(* Logix 5000 project; controller QW361 vendor 1 type 14 code 107 rev 32.11; software revision 32.00; part 19 of 20 *)
(* tags used below, declared in another part *)
   ALM_ACK : BOOL;   // Alarm acknowledge
   alm_pwrup_done : BOOL;
   ALM_RESET : BOOL;   // Alarm reset
   ALM_TEST : BOOL;   // Alarm test
   analogfb_pwrup_done : BOOL;
   ATSFLT : ALM;   // ATS fault
   ATSGEN : ALM;   // ATS in generator
   BAND_B01_MAXSPD_LVL : REAL;   // Band 1 maximum speed level
   BAND_B01_MINSPD_LVL : REAL;   // Band 1 minimum speed level
   BAND_B01_START : REAL;   // Wet well level to start lead pump
   BAND_B01_STOP : REAL;   // Wet well level to stop lead pump
   BAND_B02_MAXSPD_LVL : REAL;   // band 2 maximum speed level
   BAND_B02_MINSPD_LVL : REAL;   // band 2 minimum speed level
   BAND_B02_START : REAL;   // Wet well level to start lag pump
   BAND_B02_STOP : REAL;   // Wet well level to stop lag pump
   BAND_CURRENT : DINT;   // Current band
   CRP : ALM;   // Control power failure
   DG1 : MOTOR;   // Diesel generator
   DG1_FL : ALM;   // Diesel generator fault alarm
   DG1BAT : ALM;   // Battery low / fail
   DG1LSL1 : ALM;   // Low fuel
   DG1LSL2 : ALM;   // Low oil
   DG1RUN : ALM;   // Diesel generator running
   Dialer : BOOL[256];
   DIALOUT_ON : BOOL;
   digitalnf_pwrup_done : BOOL;
   duty_pwrup_done : BOOL;
   FIT001 : PRANALOG;   // Station discharge flow
   FIT001_CA : ALM;   // Station discharge flow calibrate mode alarm
   FIT001_FL : ALM;   // Station discharge flow sensor fail alarm
   FIT001_hh : ALM;   // Station discharge flow high high alarm
   FIT001_hi : ALM;   // Station discharge flow high alarm
   FIT001_ll : ALM;   // Station discharge flow low low alarm
   FIT001_lo : ALM;   // Station discharge flow low alarm
   FROM_QW360 : COMMBLOCK;
   FunctionBlock_Cycle_Time : REAL;   // Main Task Cycle Time in mseconds
   HardwareFault : BOOL;   // System hardware fault
   HMI_time : DateTime;
   HMI_time_set : BOOL;
   Last_Minute : DINT;
   LIT001 : PRANALOG;   // Wet well level
   LIT001_CA : ALM;   // Wet well level calibrate mode alarm
   LIT001_FL : ALM;   // Wet well level sensor fail alarm
   LIT001_hh : ALM;   // Wet well level high high alarm
   LIT001_hi : ALM;   // Wet well level high alarm
   LIT001_ll : ALM;   // Wet well level low low alarm
   LIT001_lo : ALM;   // Wet well level low alarm
   LSH001 : ALM;   // Station high float
   LSH002 : ALM;   // Station hihi float
   main_comm_pwrup_done : BOOL;
   MainTask_Cycle_Time : REAL;   // Main Task Cycle Time in mseconds
   motor_pwrup_done : BOOL;
   P001 : MOTOR;   // Raw sewage pump 1
   P001_FL : ALM;   // Raw sewage pump 1 fault alarm
   P001_LK : BOOL;   // Raw sewage pump 1 leak
   P001_OL : BOOL;   // Raw sewage pump 1 overload
   P001_TMP : BOOL;   // Raw sewage pump 1 temp
   P001SP : ANALOGFB;   // Raw sewage pump 1 speed
   P001SP_FL : ALM;   // Raw sewage pump 1 speed control fail alarm
   P002 : MOTOR;   // Raw sewage pump 2
   P002_FL : ALM;   // Raw sewage pump 2 fault alarm
   P002_LK : BOOL;   // Raw sewage pump 2 leak
   P002_OL : BOOL;   // Raw sewage pump 2 overload
   P002_TMP : BOOL;   // Raw sewage pump 2 temp
   P002SP : ANALOGFB;   // Raw sewage pump 2 speed
   P002SP_FL : ALM;   // Raw sewage pump 2 speed control fail alarm
   P00x : DUTY;   // Raw sewage pump duty
   P00xXA1 : ALM;   // Single raw sewage pump unavailable
   P00xXA2 : ALM;   // Multiple raw sewage pump unavailable
   pid_pwrup_done : BOOL;
   pranalog_pwrup_done : BOOL;
   pwrdown_time : DINT;
   report_pwrup_done : BOOL;
   sequence_pwrup_done : BOOL;
   SoftwareFault : BOOL;   // System software fault
   TO_QW360 : COMMBLOCK;
   valve_pwrup_done : BOOL;
   WALLCLOCK : DateTime;   // Global date / time
   WALLCLOCK_lock : BOOL;
   Watchdog_Relay : BOOL;
   XAFLOAT : ALM;   // Station in float mode
   XAHWARE : ALM;   // PLC hardware fault
   XASWARE : ALM;   // PLC software fault

PROGRAM AlmProgram   (* main routine Alms *)
VAR
   alm : ALM := (enmn := 1, enau := 1, alarm_tonr.TimerEnable := 1, alarm_tonr.Reset := 1);
   bit_num : DINT := 256;
   channel_num : DINT := 257;
   Controller_Status : DINT := 12640;
   Dint_Bit : DINT := 31;
   Dint_Word : DINT := 7;
   fail_pending : BOOL;
   Faulty_Modules : DINT := 3;
   latched_alarm : BOOL;
   num_channels : DINT := 256;
   temp_array : BOOL[256];
END_VAR

ROUTINE AlmRoutine   (* structured text *)
   SBR(alm);
   
   (* Alm function block *)
   
   (* Does all control processing for alarms *)
   
   (* Calling parameters: *)
   (*     alm : ALM *)
   
   (* Globals used: *)
   
   (* Globals changed: *)
   (*     fail_pending *)
   
   (*-------------------------------------------------------------------------------------------------------------------------------------------------*)
   //alm.enmn := 1;
   
   (* Load fault time with preset value *)
   alm.alarm_tonr.PRE := alm.dlay * 1000;
   alm.alarm_tonr.TimerEnable := 1;
   
   (* handle the alarms and events outputs *)
   
   (* check for previously latched alarms *)
   latched_alarm := alm.alarm AND alm.latch AND NOT alm.reset;
   
   (* calculate the fail pending *)
   IF
           NOT alm.enau
       OR
           NOT alm.enmn
       OR
           NOT alm.raw AND NOT latched_alarm
   
   THEN
       fail_pending := 0;
   
   ELSE
       fail_pending := 1;
   END_IF;
   
   (* time the fail pending *)
   alm.alarm_tonr.Reset := NOT fail_pending;
   TONR(alm.alarm_tonr);
   
   (* get the output *)
   alm.alarm := alm.alarm_tonr.DN;
   
   (* turn on the alarm channel if this is in alarm *)
   IF alm.alarm AND alm.chan > 0 AND alm.chan <= num_channels THEN
       temp_array[alm.chan - 1] := 1;
   END_IF;
   
   (* reset mometaries *)
   IF alm.reset THEN alm.reset := 0; END_IF;
   
   RET(alm);
   
END_ROUTINE

ROUTINE Alms   (* structured text *)
   (* Alm processing program *)
   
   (* Does all basic processing for all alms by calling the alm function block for each *)
   
   (* Globals used: *)
   
   (* Globals changed: *)
   (*     alm_pwrup_done *)
   
   (*-------------------------------------------------------------------------------------------------------------------------------------------------*)
   
   
   (* clear the channel array *)
   
   (* get the size of the channel array *)
   num_channels := 256;
   
   (* now clear the entire array *)
   FOR channel_num := 1 TO num_channels DO
       temp_array[channel_num - 1] := 0;
   END_FOR;
   
   
   (* get the fault records *)
   GSV( MODULE, , ledstatus, Faulty_Modules );
   GSV(CONTROLLERDEVICE, , STATUS, Controller_Status );
   
   (* hardware fault if the IO light is neither solid on or off OR major fault or minor fault unrecoverable *)
   HardwareFault := ((Faulty_Modules <> 3) AND (Faulty_Modules <> 0)) OR ((Controller_Status AND 16#F00) <> 0);
   
   (* software fault if the unit is not in run mode (includes unrecoverable faults) *)
   SoftwareFault := (Controller_Status AND 16#FF) <> 16#60;
   
   
   (************ insert alms here ***************)
   
   (* 1.  Call the discrete alarms *)
   JSR (Discretes);
   
   (* 2.  Call the motor alarms *)
   JSR (Motors);
   
   (* 3.  Call the valve alarms *)
   JSR (Valves);
   
   (* 4.  Call the pranalog alarms *)
   JSR (Pranalogs);
   
   (* 5.  Call the Analogfb alarms *)
   JSR (Analogfbs);
   
   
   (* XAHWARE PLC Hardware fault *)
   
   (* process the inputs *)
   XAHWARE.raw := HardwareFault;
   XAHWARE.enau := 1;
   
   (* process the alarm *)
   JSR( AlmRoutine, 1, XAHWARE, XAHWARE );
   
   
   (* XASWARE PLC Software fault *)
   
   (* process the inputs *)
   XASWARE.raw := SoftwareFault;
   XASWARE.enau := 1;
   
   (* process the alarm *)
   JSR( AlmRoutine, 1, XASWARE, XASWARE );
   
   
   (* now copy the results from the temp array to the permanent array *)
   DIALOUT_ON := 0;
   FOR bit_num := 0 to 255 DO
   	Dint_Word := bit_num / 32;
   	Dint_Bit := bit_num - (Dint_Word * 32);
   	Dialer[bit_num] := temp_array[bit_num];
   	TO_QW360.ALMDINTS[Dint_Word].[Dint_Bit] := temp_array[bit_num];
   	IF Dialer[bit_num] THEN
   		DIALOUT_ON := 1;
   	END_IF;
   END_FOR;
   
   
   (* flag that powerup is done *)
   alm_pwrup_done := 1;
   
   
END_ROUTINE

ROUTINE Analogfbs   (* structured text *)
   (* P001SP_FL Raw sewage pump 1 speed control fail alarm *)
   
   (* process the inputs *)
   P001SP_FL.raw := P001SP_FL.raw;
   P001SP_FL.enau := 1;
   
   (* process the alarm *)
   JSR( AlmRoutine, 1, P001SP_FL, P001SP_FL );
   
   
   (* P002SP_FL Raw sewage pump 2 speed control fail alarm *)
   
   (* process the inputs *)
   P002SP_FL.raw := P002SP_FL.raw;
   P002SP_FL.enau := 1;
   
   (* process the alarm *)
   JSR( AlmRoutine, 1, P002SP_FL, P002SP_FL );
END_ROUTINE

ROUTINE Discretes   (* structured text *)
   
   (* CRP Control power failure *)
   
   (* process the inputs *)
   CRP.raw := CRP.raw;
   CRP.enau := 1;
   
   (* process the alarm *)
   JSR( AlmRoutine, 1, CRP, CRP );
   
   
   (* LS001 Station high float *)
   
   (* process the inputs *)
   LSH001.raw := LSH001.raw;
   LSH001.enau := 1;
   
   (* process the alarm *)
   JSR( AlmRoutine, 1, LSH001, LSH001 );
   
   
   (* LS002 Station hihi float *)
   
   (* process the inputs *)
   LSH002.raw := LSH002.raw;
   LSH002.enau := 1;
   
   (* process the alarm *)
   JSR( AlmRoutine, 1, LSH002, LSH002 );
   
   
   (* XAFLOAT Station in float mode *)
   
   (* process the inputs *)
   XAFLOAT.raw := XAFLOAT.raw;
   XAFLOAT.enau := 1;
   
   (* process the alarm *)
   JSR( AlmRoutine, 1, XAFLOAT, XAFLOAT );
   
   
   (* DG1LSL1 Low fuel *)
   
   (* process the inputs *)
   DG1LSL1.raw := DG1LSL1.raw;
   DG1LSL1.enau := 1;
   
   (* process the alarm *)
   JSR( AlmRoutine, 1, DG1LSL1, DG1LSL1 );
   
   
   (* DG1LSL2 Low oil *)
   
   (* process the inputs *)
   DG1LSL2.raw := DG1LSL2.raw;
   DG1LSL2.enau := 1;
   
   (* process the alarm *)
   JSR( AlmRoutine, 1, DG1LSL2, DG1LSL2 );
   
   
   (* DG1BAT Battery low / fail *)
   
   (* process the inputs *)
   DG1BAT.raw := DG1BAT.raw;
   DG1BAT.enau := 1;
   
   (* process the alarm *)
   JSR( AlmRoutine, 1, DG1BAT, DG1BAT );
   
   
   (* DG1RUN Diesel generator running *)
   
   (* process the inputs *)
   DG1RUN.raw := DG1.run_sts;
   DG1RUN.enau := 1;
   
   (* process the alarm *)
   JSR( AlmRoutine, 1, DG1RUN, DG1RUN );
   
   
   (* ATSGEN ATS in generator *)
   
   (* process the inputs *)
   ATSGEN.raw := ATSGEN.raw;
   ATSGEN.enau := 1;
   
   (* process the alarm *)
   JSR( AlmRoutine, 1, ATSGEN, ATSGEN );
   
   
   (* ATSFLT ATS fault *)
   
   (* process the inputs *)
   ATSFLT.raw := ATSFLT.raw;
   ATSFLT.enau := 1;
   
   (* process the alarm *)
   JSR( AlmRoutine, 1, ATSFLT, ATSFLT );
   
   
   (* P00xXA1 Single raw sewage pump unavailable *)
   
   (* process the inputs *)
   P00xXA1.raw := P00xXA1.raw;
   P00xXA1.enau := 1;
   
   (* process the alarm *)
   JSR( AlmRoutine, 1, P00xXA1, P00xXA1 );
   
   
   (* P00xXA2 Multiple raw sewage pump unavailable *)
   
   (* process the inputs *)
   P00xXA2.raw := P00xXA2.raw;
   P00xXA2.enau := 1;
   
   (* process the alarm *)
   JSR( AlmRoutine, 1, P00xXA2, P00xXA2 );
   
   
   
   
END_ROUTINE

ROUTINE Motors   (* structured text *)
   (* P001_FL Raw sewage pump 1 fault alarm *)
   
   (* process the inputs *)
   P001_FL.raw := P001_FL.raw;
   P001_FL.enau := 1;
   
   (* process the alarm *)
   JSR( AlmRoutine, 1, P001_FL, P001_FL );
   
   
   (* P002_FL Raw sewage pump 2 fault alarm *)
   
   (* process the inputs *)
   P002_FL.raw := P002_FL.raw;
   P002_FL.enau := 1;
   
   (* process the alarm *)
   JSR( AlmRoutine, 1, P002_FL, P002_FL );
   
   
   (* DG1_FL Diesel generator fault alarm *)
   
   (* process the inputs *)
   DG1_FL.raw := DG1_FL.raw;
   DG1_FL.enau := 1;
   
   (* process the alarm *)
   JSR( AlmRoutine, 1, DG1_FL, DG1_FL );
END_ROUTINE

ROUTINE Pranalogs   (* structured text *)
   (* LIT001_hi Wet well level high alarm *)
   
   (* process the inputs *)
   LIT001_hi.raw := LIT001_hi.raw;
   LIT001_hi.enau := 1;
   
   (* process the alarm *)
   JSR( AlmRoutine, 1, LIT001_hi, LIT001_hi );
   
   
   (* LIT001_lo Wet well level low alarm *)
   
   (* process the inputs *)
   LIT001_lo.raw := LIT001_lo.raw;
   LIT001_lo.enau := 1;
   
   (* process the alarm *)
   JSR( AlmRoutine, 1, LIT001_lo, LIT001_lo );
   
   
   (* LIT001_hh Wet well level high high alarm *)
   
   (* process the inputs *)
   LIT001_hh.raw := LIT001_hh.raw;
   LIT001_hh.enau := 1;
   
   (* process the alarm *)
   JSR( AlmRoutine, 1, LIT001_hh, LIT001_hh );
   
   
   (* LIT001_ll Wet well level low low alarm *)
   
   (* process the inputs *)
   LIT001_ll.raw := LIT001_ll.raw;
   LIT001_ll.enau := 1;
   
   (* process the alarm *)
   JSR( AlmRoutine, 1, LIT001_ll, LIT001_ll );
   
   
   (* LIT001_CA Wet well level calibrate mode alarm *)
   
   (* process the inputs *)
   LIT001_CA.raw := LIT001_CA.raw;
   LIT001_CA.enau := 1;
   
   (* process the alarm *)
   JSR( AlmRoutine, 1, LIT001_CA, LIT001_CA );
   
   
   (* LIT001_FL Wet well level sensor fail alarm *)
   
   (* process the inputs *)
   LIT001_FL.raw := LIT001_FL.raw;
   LIT001_FL.enau := 1;
   
   (* process the alarm *)
   JSR( AlmRoutine, 1, LIT001_FL, LIT001_FL );
   
   
   (* FIT001_hi Station discharge flow high alarm *)
   
   (* process the inputs *)
   FIT001_hi.raw := FIT001_hi.raw;
   FIT001_hi.enau := 1;
   
   (* process the alarm *)
   JSR( AlmRoutine, 1, FIT001_hi, FIT001_hi );
   
   
   (* FIT001_lo Station discharge flow low alarm *)
   
   (* process the inputs *)
   FIT001_lo.raw := FIT001_lo.raw;
   FIT001_lo.enau := 1;
   
   (* process the alarm *)
   JSR( AlmRoutine, 1, FIT001_lo, FIT001_lo );
   
   
   (* FIT001_hh Station discharge flow high high alarm *)
   
   (* process the inputs *)
   FIT001_hh.raw := FIT001_hh.raw;
   FIT001_hh.enau := 1;
   
   (* process the alarm *)
   JSR( AlmRoutine, 1, FIT001_hh, FIT001_hh );
   
   
   (* FIT001_ll Station discharge flow low low alarm *)
   
   (* process the inputs *)
   FIT001_ll.raw := FIT001_ll.raw;
   FIT001_ll.enau := 1;
   
   (* process the alarm *)
   JSR( AlmRoutine, 1, FIT001_ll, FIT001_ll );
   
   
   (* FIT001_CA Station discharge flow calibrate mode alarm *)
   
   (* process the inputs *)
   FIT001_CA.raw := FIT001_CA.raw;
   FIT001_CA.enau := 1;
   
   (* process the alarm *)
   JSR( AlmRoutine, 1, FIT001_CA, FIT001_CA );
   
   
   (* FIT001_FL Station discharge flow sensor fail alarm *)
   
   (* process the inputs *)
   FIT001_FL.raw := FIT001_FL.raw;
   FIT001_FL.enau := 1;
   
   (* process the alarm *)
   JSR( AlmRoutine, 1, FIT001_FL, FIT001_FL );
   
END_ROUTINE

ROUTINE Valves   (* structured text *)
   
END_ROUTINE
END_PROGRAM

PROGRAM AnalogfbProgram   (* main routine Analogfbs *)
VAR
   analogfb : ANALOGFB := (remote := 1, permit := 1, fail_tonr.TimerEnable := 1, fail_tonr.Reset := 1);
   fail_pending : BOOL;
   pwrup_dlayd : FBD_TIMER := (TimerEnable := 1, PRE := 10000, ACC := 10000, EN := 1, DN := 1);
END_VAR

ROUTINE AnalogfbRoutine   (* structured text *)
   SBR(analogfb);
   
   (* Analogfb function block *)
   
   (* Does all control processing for analog devices with feedback *)
   
   (* Calling parameters: *)
   (*     analogfb : ANALOGFB *)
   
   (* Globals used: *)
   (*     pwrup_dlayd *)
   
   (* Globals changed: *)
   (*     fail_pending *)
   
   (*-------------------------------------------------------------------------------------------------------------------------------------------------*)
   
   
   (* handle the failure logic first *)
   
   (* calculate the fail pending *)
   IF
           NOT analogfb.remote
       OR
   	    ( ABS( analogfb.out - analogfb.feedback ) <= 5.0 )
   	OR
   	    NOT pwrup_dlayd.DN
   THEN
       fail_pending := 0;
   ELSE
       fail_pending := 1;
   END_IF;
   
   (* time the fail pending *)
   analogfb.fail_tonr.PRE := analogfb.fail_dlay * 1000;
   analogfb.fail_tonr.TimerEnable := 1;
   analogfb.fail_tonr.Reset := NOT fail_pending;
   tonr(analogfb.fail_tonr);
   
   (* calculate the fail and clear if we're not in remote or we just powered up *)
   analogfb.fail := ( analogfb.fail AND ( NOT analogfb.fail_reset AND analogfb.remote AND pwrup_dlayd.DN ) ) OR analogfb.fail_tonr.DN;
   
   
   (* make the feedback *)
   IF analogfb.feedback_raw < 2 THEN
   	analogfb.feedback := 0;
   ELSIF analogfb.feedback_raw > 98 THEN
   	analogfb.feedback := 100;
   ELSE
   	analogfb.feedback := analogfb.feedback_raw;
   END_IF;
   
   
   (* handle the analog fb outputs *)
   
   (* if we're not permitted to control or not in remote or just powered up, set output to current feedback *)
   IF NOT analogfb.permit OR NOT analogfb.remote OR NOT pwrup_dlayd.DN THEN
   	analogfb.out := analogfb.feedback;
   
   (* if we're not in auto, set the output to the manual setpoint and track with the auto setpoint *)
   ELSIF NOT analogfb.auto THEN
   	analogfb.out := analogfb.out_man;
   
   (* otherwise, set the output to the auto setpoint and track with the manual setpoint*)
   ELSE
   	analogfb.out := analogfb.out_auto;
   END_IF;
   
   (* make sure both setpoints track *)
   analogfb.out_man := analogfb.out;
   analogfb.out_auto:= analogfb.out;
   
   
   (* process the momentary resets *)
   
   (* set the momentary resets equal to the current state *)
   IF analogfb.fail_reset THEN analogfb.fail_reset := 0; END_IF;
   
   RET(analogfb);
END_ROUTINE

ROUTINE Analogfbs   (* structured text *)
   (* Analogfb processing program *)
   
   (* Does all basic processing for all analogfbs by setting up inputs then calling the analogfb function block for each *)
   
   (* Globals used: *)
   
   (* Globals changed: *)
   (*     analogfb_pwrup_done *)
   (*     pwrup_dlayd *)
   (*     each analogfb *)
   
   (*-------------------------------------------------------------------------------------------------------------------------------------------------*)
   
   
   (* use a TONR to delay ac power recovery *)
   
   pwrup_dlayd.Reset := not analogfb_pwrup_done;
   TONR(pwrup_dlayd);
   
   
   (* process each analogfb as follows: (note these comments are only shown here for brevity) *)
   (*     1. set up inputs (specific to each analogfb and commented *)
   (*     2. call the analogfb processing function block *)
   (*     3. clear the momentary inputs if they were on *)
   (*     4. get the outputs *)
   
   
   (************ insert analogfbs here ***************)
   
   
   (* P001SP Raw sewage pump 1 speed *)
   
   (* set up the inputs *)
   P001SP.remote := 1;
   P001SP.permit := 1;
   P001SP.feedback_raw := P001SP.out;
   
   (* process the analog with feedback and reset the momentaries *)
   JSR( AnalogfbRoutine, 1, P001SP, P001SP );
   P001SP_FL.raw := P001SP.fail;
   
   
   (* P002SP Raw sewage pump 2 speed *)
   
   (* set up the inputs *)
   P002SP.remote := 1;
   P002SP.permit := 1;
   P002SP.feedback_raw := P002SP.out;
   
   (* process the analog with feedback and reset the momentaries *)
   JSR( AnalogfbRoutine, 1, P002SP, P002SP );
   P002SP_FL.raw := P002SP.fail;
   
   
   
   (* flag that powerup is done *)
   analogfb_pwrup_done := 1;
   
END_ROUTINE
END_PROGRAM

PROGRAM Communication   (* main routine Main_Comm *)
VAR
   bit_num : DINT := 256;
   WD_in : DINT := 6947;
   WD_out : DINT := 6947;
END_VAR

ROUTINE Main_Comm   (* structured text *)
   (* Message routine for communication from PLC to PLC *)
   
   (* Globals used: *)
   
   (* Globals changed: *)
   
   (*-------------------------------------------------------------------------------------------------------------------------------------------------*)
   
   
   (************ insert comm stuff here ***************)
   (* send data to Youngs Cove WWTP *)
   
   (* Plant PLC COMMS *)
   (* Monitor / Control the WatchDog from QW360.  This side is the slave side, we recieve a watchdog
   	number and loop it back.  If the number we read fails to change then communications has failed.
   	Once we get an new number it's ok. *)
   IF TO_QW360.WATCHDOG <> FROM_QW360.WATCHDOG THEN
   //	XA_LLCOMM.Raw := 0;
   	TO_QW360.WATCHDOG := FROM_QW360.WATCHDOG;
   ELSE
   //	XA_LLCOMM.Raw := 1;
   END_IF;
   
   
   (* Output Block to Plant PLC *)
   	(* Watchdog - done above *)
   	(* BOOLS *)
   	TO_QW360.BOOLS[0] := DIALOUT_ON; //dialer zone is active
   
   	(* INTEGERS *)
   	TO_QW360.DINTS[0] := 0;
   
   	(* REALS *)
   	TO_QW360.REALS[0] := LIT001.value;
   	TO_QW360.REALS[1] := FIT001.value;
   
   
   
   
   (* Input Block From Tower PLC *)
   	(* Watchdog - done above *)
   	(* BOOLS *)
   // := FROM_QW360.BOOLS[0];
   
   	(* INTEGERS *)
   // := FROM_QW360.DINTS[0];
   
   	(* REALS *)
   // := FROM_QW360.REALS[0]; //
   
   	(* ALARMS *)
   // Used directly in Alms subroutine;
   
   
   (* flag that powerup is done *)
   main_comm_pwrup_done := 1;
   
END_ROUTINE
END_PROGRAM

PROGRAM CycleTime   (* main routine MainRoutine *)
VAR
   cycle_timer1 : FBD_TIMER := (TimerEnable := 1, Reset := 1, ACC := 500, EN := 1, DN := 1);
   cycle_timer2 : FBD_TIMER := (TimerEnable := 1, EN := 1, TT := 1);
   cycle_timer3 : FBD_TIMER := (TimerEnable := 1);
   DATETIME_TEMP : DateTime := (Year := 2022, Month := 5, Day := 3, Hour := 16, Minute := 29, Second := 58, Microsecond := 621793, DayOfWeek := 2, DST_ON := 1);
   DOW_Century : DINT := 20;   // Century or upper two digits from the year
   DOW_Day : DINT := 3;   // Day of the Month 1-31
   DOW_Month : DINT := 3;   // Month 1 = March, 10=december, 11=Jan and 12=Feb
   DOW_Output : DINT := 2;   // Day of Week 0 = Sun, 1=Mon, 2=Tues, 3=Wed, 4=Thur, 5=Fri, 6=Sat
   DOW_Temp00 : REAL := 20.22;   // Intermediate Math Value
   DOW_Temp01 : REAL := 7.7999997;   // Intermediate Math Value
   DOW_Temp02 : REAL := 7.600001;   // Intermediate Math Value
   DOW_Temp03 : DINT := 7;   // Intermediate Math Value
   DOW_Temp04 : DINT := 40;   // Intermediate Math Value
   DOW_Temp05 : REAL := 5.5;   // Intermediate Math Value
   DOW_Temp06 : DINT := 5;   // Intermediate Math Value
   DOW_Temp07 : REAL := 5.0;   // Intermediate Math Value
   DOW_Temp08 : DINT := 5;   // Intermediate Math Value
   DOW_Temp09 : REAL := 10.0;   // Intermediate Math Value
   DOW_Temp10 : REAL := -30.0;   // Intermediate Math Value
   DOW_Temp11 : REAL := -8.0;   // Intermediate Math Value
   DOW_Temp12 : REAL := -3.0;   // Intermediate Math Value
   DOW_Temp13 : REAL := 2.0;   // Intermediate Math Value
   DOW_Temp14 : REAL := 2.0;   // Intermediate Math Value
   DOW_Temp15 : REAL := 2.0;   // Intermediate Math Value
   DOW_Year : DINT := 22;   // Year within the century or last two digits in year
END_VAR

ROUTINE CycleTime   (* structured text *)
   (* determine elapsed time of this task since last execution using three timers *)
   
   (* get the three timers elapsed time *)
   (* note one timer is resetting and the other two are timing *)
   TONR(cycle_timer1);
   TONR(cycle_timer2);
   TONR(cycle_timer3);
   
   (* of course, grab the output from the timer that was reset two cycles ago and add in any powerdown time *)
   IF cycle_timer1.Reset THEN
       MainTask_Cycle_Time := cycle_timer2.ACC + pwrdown_time;
   	cycle_timer1.Reset := 0;
   	cycle_timer2.Reset := 1;
   	cycle_timer3.Reset := 0;
   ELSIF cycle_timer2.Reset THEN
       MainTask_Cycle_Time := cycle_timer3.ACC + pwrdown_time;
   	cycle_timer1.Reset := 0;
   	cycle_timer2.Reset := 0;
   	cycle_timer3.Reset := 1;
   ELSE
       MainTask_Cycle_Time := cycle_timer1.ACC + pwrdown_time;
   	cycle_timer1.Reset := 1;
   	cycle_timer2.Reset := 0;
   	cycle_timer3.Reset := 0;
   END_IF;
   
   
   
   
END_ROUTINE

ROUTINE DayOfWeek   (* ladder *)
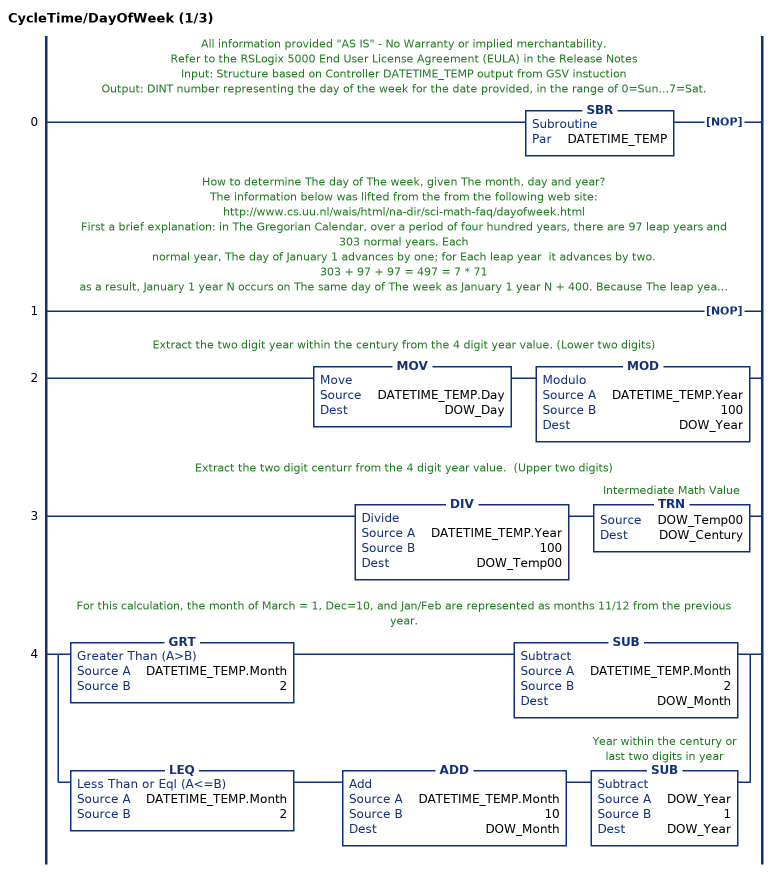
   // All information provided "AS IS" - No Warranty or implied merchantability.
   // Refer to the RSLogix 5000 End User License Agreement (EULA) in the Release Notes
   // Input: Structure based on Controller DATETIME_TEMP output from GSV instuction
   // Output: DINT number representing the day of the week for the date provided, in the range of 0=Sun...7=Sat.
   0: SBR(DATETIME_TEMP)NOP();
   // How to determine The day of The week, given The month, day and year?
   // The information below was lifted from the from the following web site: http://www.cs.uu.nl/wais/html/na-dir/sci-math-faq/dayofweek.html
   //    First a brief explanation: in The Gregorian Calendar, over a period of four hundred years, there are 97 leap years and 303 normal years. Each
   //  normal year, The day of January 1 advances by one; for Each leap year  it advances by two.
   //    303 + 97 + 97 = 497 = 7 * 71
   //    as a result, January 1 year N occurs on The same day of The week as January 1 year N + 400. Because The leap year pattern also recurs with a four hundred year cycle, a simple table of four hundred elements, and single modulus, suffices to determine The day of The week (in The
   //    Gregorian Calendar), and does it much faster than all The other algorithms proposed. also, Each element takes (in principle) only three bits; The entire table thus takes only 1200 bits; on many computers this will be less than The instructions to do all The complicated calculations proposed or The other algorithms.
   //    Incidental Note: Because 7 does not Divide 400, January 1 occurs more frequently on some days than others! Trick your friends! in a cycle of 400 years, January 1 and March 1 occur on The following days with The following frequencies:
   //            Sun      Mon     Tue     Wed     Thu     Fri     Sat
   //     Jan 1: 58       56      58      57      57      58      56
   //     Mar 1: 58       56      58      56      58      57      57
   //    Of interest is that (contrary to most initial guesses) The occurrence is not maximally flat.
   // In The Mathematical Gazette, vol. 53,, pp.127-129, it is shown that The 13th of The month is more likely to be a Friday than any other day.The author is a 13 year old S.R.Baxter.
   //    The Gregorian Calendar was introduced in 1582 in parts of Europe; it was adopted in 1752 in Great Britain and its colonies, and on various dates in other countries. it replaced The Julian Calendar which has a four-year cycle of leap years; after four years January 1 has advanced by five days. Since 5 is relatively prime to 7, a table of 4 * 7 = 28 elements is necessary for The Julian Calendar.
   //    there is still a 3 day over 10,000 years error which The Gregorian Calendar does not take into account. At some Time such a correction will have to be done but your software will probably not last that long!
   //    Here is a standard method suitable for mental computation:
   //     1. take The last two digits of The year.
   //     2. Divide by 4, discarding any fraction.
   //     3. Add The day of The month.
   //     4. Add The month'S key value: JFM AMJ JAS OND 144 025 036 146
   //     5. Subtract 1 for January or February of a leap year.
   //     6. For a Gregorian Date, Add 0 for 1900'S, 6 for 2000'S, 4 for 1700'S, 2 for 1800'S; for other years, Add or Subtract multiples of 400.
   //     7. For a Julian Date, Add 1 for 1700'S, and 1 for every additional century you go back.
   //     8. Add The last two digits of The year.
   //     9. Divide by 7 and take The remainder.
   //    Now 1 is Sunday, The First day of The week, 2 is Monday, and so on.
   //    The following formula, which is for The Gregorian Calendar only, may be more convenient for computer programming. Note that in some programming languages The remainder operation can yield a negative result if given a negative operand, so mod 7 may not translate to a simple remainder.
   //    W = (k + floor(2.6m - 0.2) - 2C + Y + floor(Y/4) + floor(C/4)) mod 7
   //    where floor() denotes The integer floor function [This is TRN() in Logix],
   // k is day (1 to 31)
   //  m is month (1 = March, ..., 10 = December, 11 = Jan, 12 = Feb) Treat Jan & Feb as months of The preceding year
   //    C is century (1987 has C = 19)
   //    Y is year (1987 has Y = 87 except Y = 86 for Jan & Feb)
   //    W is week day (0 = Sunday, ..., 6 = Saturday)
   //    Here The century and 400 year corrections are built into The formula. The floor(2.6m - 0.2) term relates to The repetitive pattern that The 30-day months show when March is taken as The First month.
   //    The following short C program works for a restricted range, it returns 0 for Monday, 1 for Tuesday, etc.
   // dow(m,d,Y){Y-=m<3;return(Y+Y/4-Y/100+Y/400+"-bed=pen+mad."[m]+d)%7;}
   //    The program appeared was posted by sakamoto@sm.sony.co.jp (Tomohiko sakamoto) on comp.lang.c on March 10th, 1993.
   //    a good mnemonic rule to help on The computation of The day of The week is as follows. in any given year The following days come on The same day of The week: 4/4, 6/6, 8/8, 10/10, 12/12  to remember The next four, remember that I work from 9-5 At a 7-11 so 9/5, 5/9, 7/11, 11/7 and The last day of Feb.
   //    "in 1995 they come on Tuesday. every year this advances one other than leap-years which advance 2. Therefore for 1996 The day will be Thursday, and for 1997 it will be Friday. Therefore ordinarily every 4 years it advances 5 days. there is a minor correction for The century Since The century is a leap year iff The century is divisible by 4. Therefore 2000 is a leap year, but 1900, 1800, and 1700 were not."
   //    Even ignoring The pattern over for a period of years this is still useful Since you can generally figure out what day of The week a given Date is  on faster than someone else can look it up with a calender if The calender is not right there. (a useful skill that.)
   //  References:
   //    Winning Ways for your Mathematical plays. Elwyn R. Berlekamp, John H.  Conway, and Richard k. Guy London ; Toronto : Academic Press, 1982.
   //    Mathematical Carnival. Martin Gardner. New York : Knopf, c1975.
   //    Elementary Number Theory and its applications. Kenneth Rosen. Reading,  Mass. ; Don Mills, Ont. : Addison-Wesley Pub. Co., c1993. p. 156.
   //    Michael Keith and Tom Craver. The Ultimate Perpetual Calendar? Journal of Recreational Mathematics, 22:4, pp. 280-282, 19
   1: NOP();
   // Extract the two digit year within the century from the 4 digit year value. (Lower two digits)
   2: MOV(DATETIME_TEMP.Day,DOW_Day)MOD(DATETIME_TEMP.Year,100,DOW_Year);
   // Extract the two digit centurr from the 4 digit year value.  (Upper two digits)
   3: DIV(DATETIME_TEMP.Year,100,DOW_Temp00)TRN(DOW_Temp00,DOW_Century);
   // For this calculation, the month of March = 1, Dec=10, and Jan/Feb are represented as months 11/12 from the previous year.
   4: [GRT(DATETIME_TEMP.Month,2) SUB(DATETIME_TEMP.Month,2,DOW_Month) ,LEQ(DATETIME_TEMP.Month,2) ADD(DATETIME_TEMP.Month,10,DOW_Month) SUB(DOW_Year,1,DOW_Year) ];
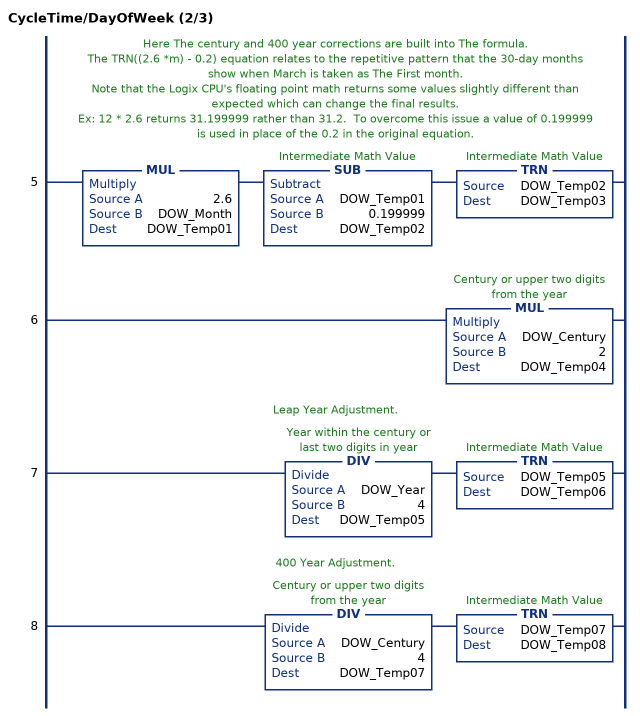
   // Here The century and 400 year corrections are built into The formula.
   // The TRN((2.6 *m) - 0.2) equation relates to the repetitive pattern that the 30-day months show when March is taken as The First month.
   // Note that the Logix CPU's floating point math returns some values slightly different than expected which can change the final results.
   // Ex: 12 * 2.6 returns 31.199999 rather than 31.2.  To overcome this issue a value of 0.199999 is used in place of the 0.2 in the original equation.
   5: MUL(2.6,DOW_Month,DOW_Temp01)SUB(DOW_Temp01,0.199999,DOW_Temp02)TRN(DOW_Temp02,DOW_Temp03);
   6: MUL(DOW_Century,2,DOW_Temp04);
   // Leap Year Adjustment.
   7: DIV(DOW_Year,4,DOW_Temp05)TRN(DOW_Temp05,DOW_Temp06);
   // 400 Year Adjustment.
   8: DIV(DOW_Century,4,DOW_Temp07)TRN(DOW_Temp07,DOW_Temp08);
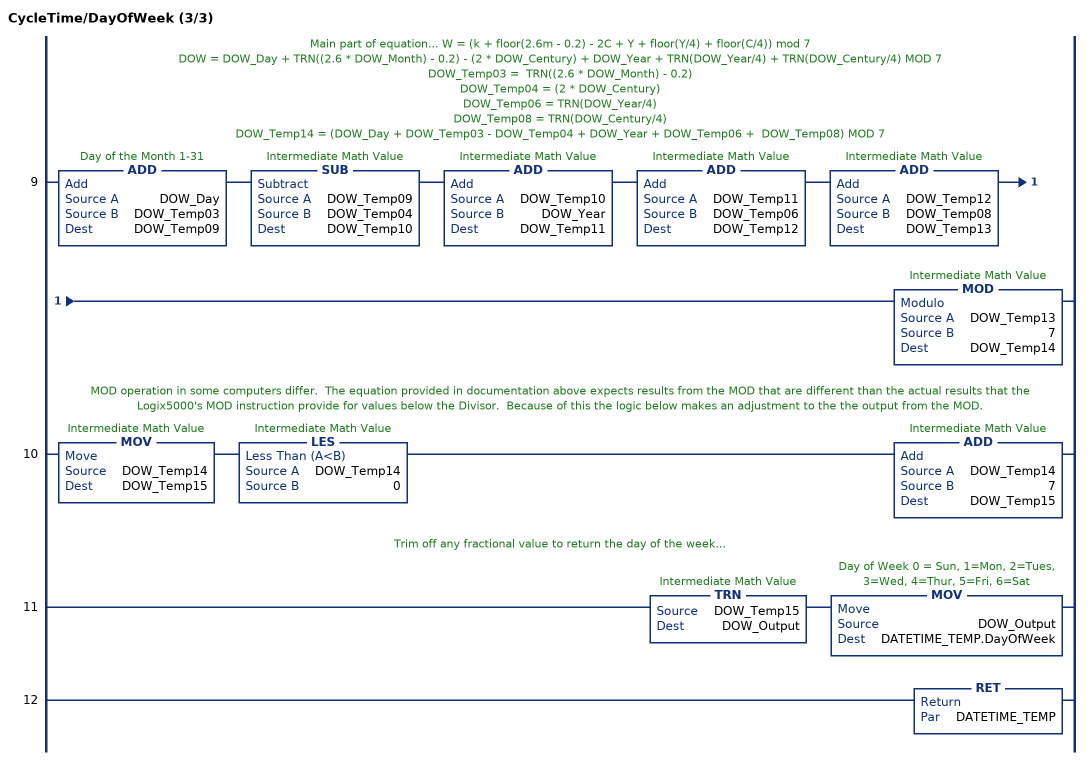
   // Main part of equation... W = (k + floor(2.6m - 0.2) - 2C + Y + floor(Y/4) + floor(C/4)) mod 7
   // DOW = DOW_Day + TRN((2.6 * DOW_Month) - 0.2) - (2 * DOW_Century) + DOW_Year + TRN(DOW_Year/4) + TRN(DOW_Century/4) MOD 7
   // DOW_Temp03 =  TRN((2.6 * DOW_Month) - 0.2)
   // DOW_Temp04 = (2 * DOW_Century)
   // DOW_Temp06 = TRN(DOW_Year/4)
   // DOW_Temp08 = TRN(DOW_Century/4)
   // DOW_Temp14 = (DOW_Day + DOW_Temp03 - DOW_Temp04 + DOW_Year + DOW_Temp06 +  DOW_Temp08) MOD 7
   9: ADD(DOW_Day,DOW_Temp03,DOW_Temp09)SUB(DOW_Temp09,DOW_Temp04,DOW_Temp10)ADD(DOW_Temp10,DOW_Year,DOW_Temp11)ADD(DOW_Temp11,DOW_Temp06,DOW_Temp12)ADD(DOW_Temp12,DOW_Temp08,DOW_Temp13)MOD(DOW_Temp13,7,DOW_Temp14);
   // MOD operation in some computers differ.  The equation provided in documentation above expects results from the MOD that are different than the actual results that the Logix5000's MOD instruction provide for values below the Divisor.  Because of this the logic below makes an adjustment to the the output from the MOD.
   10: MOV(DOW_Temp14,DOW_Temp15)LES(DOW_Temp14,0)ADD(DOW_Temp14,7,DOW_Temp15);
   // Trim off any fractional value to return the day of the week...
   11: TRN(DOW_Temp15,DOW_Output)MOV(DOW_Output,DATETIME_TEMP.DayOfWeek);
   12: RET(DATETIME_TEMP);
END_ROUTINE

ROUTINE HMI_TimeSet   (* structured text *)
   (* HMI_time_set *)
   
   (* Used to allow control of the Controller clock with operator intervention (ie SCADA) *)
   
   (* language:
     IEC 1131 Structured Text *)
   
   (* creation date:
     Dec 16, 2005 *)
   
   (* author:	Dakins Engineering Group *)
   
   (* Globals used: *)
   
   
   (* Globals changed: *)
   
   
   (*--------------------------------------------------------------------------------------------*)
   
   
   SBR();
   
   (* Set the clock if requested to *)
   IF HMI_time_set THEN
   	WALLCLOCK_lock := 1;
   	SSV( WALLCLOCKTIME, , localDateTime, HMI_time.Year );
   	WALLCLOCK.DST_ON := HMI_time.DST_ON;
   	HMI_time_set := 0;
   END_IF;
   
   RET();
   
   
END_ROUTINE

ROUTINE MainRoutine   (* structured text *)
// Handles all clock / timing functions
   (* CycleTime Program *)
   
   (* Handles all clock and timing functions  *)
   
   (* Globals used: *)
   
   (* Globals changed: *)
   
   (*-------------------------------------------------------------------------------------------------------------------------------------------------*)
   
   
   (*1.  Calculate Cycle time for use in totalizers and time counters in entire program  *)
   JSR(CycleTime);
   
   
   (*2.  Check for HMI time set *)
   JSR(HMI_TimeSet, 0);
   
   
   (*3.  Get current date/time *)
   WALLCLOCK_lock := 1;
   GSV( WALLCLOCKTIME, , localDateTime, WALLCLOCK.Year );
   
   
   (*4.  Check for Day of Week *)
   JSR(DayOfWeek,1,WALLCLOCK,WALLCLOCK);
   WALLCLOCK_lock := 0;
   
   
   (*5.  PLC Watchdog - One minute On, One minute Off ... *)
   IF WALLCLOCK.Second > 30 THEN
   	Watchdog_Relay := 0;
   	Last_Minute := WALLCLOCK.Minute;
   ELSE
   	Watchdog_Relay := 1;
   END_IF;
   
   
   
END_ROUTINE
END_PROGRAM

PROGRAM CycleTime1   (* main routine CycleTime *)
VAR
   cycle_timer1 : FBD_TIMER := (TimerEnable := 1, EN := 1, TT := 1);
   cycle_timer2 : FBD_TIMER := (TimerEnable := 1);
   cycle_timer3 : FBD_TIMER := (TimerEnable := 1, Reset := 1, ACC := 250, EN := 1, DN := 1);
END_VAR

ROUTINE CycleTime   (* structured text *)
   (* determine elapsed time of this task since last execution using three timers *)
   
   (* get the three timers elapsed time *)
   (* note one timer is resetting and the other two are timing *)
   TONR(cycle_timer1);
   TONR(cycle_timer2);
   TONR(cycle_timer3);
   
   (* of course, grab the output from the timer that was reset two cycles ago and add in any powerdown time *)
   IF cycle_timer1.Reset THEN
       FunctionBlock_Cycle_Time := cycle_timer2.ACC + pwrdown_time;
   	cycle_timer1.Reset := 0;
   	cycle_timer2.Reset := 1;
   	cycle_timer3.Reset := 0;
   ELSIF cycle_timer2.Reset THEN
       FunctionBlock_Cycle_Time := cycle_timer3.ACC + pwrdown_time;
   	cycle_timer1.Reset := 0;
   	cycle_timer2.Reset := 0;
   	cycle_timer3.Reset := 1;
   ELSE
       FunctionBlock_Cycle_Time := cycle_timer1.ACC + pwrdown_time;
   	cycle_timer1.Reset := 1;
   	cycle_timer2.Reset := 0;
   	cycle_timer3.Reset := 0;
   END_IF;
   
   
   
   
END_ROUTINE
END_PROGRAM

PROGRAM DigitalnfProgram   (* main routine Digitalnfs *)
VAR
   digitalnf : DIGITALNF;
END_VAR

ROUTINE DigitalnfRoutine   (* structured text *)
   SBR(digitalnf);
   
   (* Digitalnf function block *)
   
   (* Does all control processing for digital devices without feedback *)
   
   (* Calling parameters: *)
   (*     digitalnf : DIGITALNF *)
   
   (* Globals used: *)
   
   (* Globals changed: *)
   
   (*-------------------------------------------------------------------------------------------------------------------------------------------------*)
   
   
   (* handle the digital nf outputs *)
   
   IF NOT digitalnf.auto THEN
   	digitalnf.out := digitalnf.out_man;
   
   ELSE
   	digitalnf.out := digitalnf.out_auto;
   
   END_IF;
   
   (* make sure both outputs track *)
   digitalnf.out_man := digitalnf.out;
   digitalnf.out_auto := digitalnf.out;
   
   RET(digitalnf);
   
END_ROUTINE

ROUTINE Digitalnfs   (* structured text *)
   (* Digitalnf processing program *)
   
   (* Does all basic processing for all digitalnfs by calling the digitalnf function block for each *)
   
   (* Globals used: *)
   
   (* Globals changed: *)
   (*     digitalnf_pwrup_done *)
   
   (*-------------------------------------------------------------------------------------------------------------------------------------------------*)
   
   
   (************ insert digitalnfs here ***************)
   
   
   (* flag that powerup is done *)
   digitalnf_pwrup_done := 1;
   
END_ROUTINE
END_PROGRAM

PROGRAM DutyProgram   (* main routine Duties *)
VAR
   actual_lead_satisfied : BOOL;
   current_motor_index : DINT;
   date : DINT[7] := ([0] := 2022, [1] := 5, [2] := 3, [3] := 16, [4] := 29, [5] := 58, [6] := 878557);
   duty : DUTY := (rotate_on_stop := 1, qty_motors := 2, lead_motor := 1, motor_available := 3, hour_offset := 16920, day_offset := 705, hour_last := 16, all_motors_stopped.InputBit := 1);
   hour_current : DINT := 16;
   motor_available : DINT := 2;
   motors_required : DINT;
   motors_wanted_running : DINT := 2;
END_VAR

ROUTINE Duties   (* structured text *)
   (* Main processing program *)
   
   (* Call all Duty subroutine for equipment *)
   
   (* Globals used: *)
   
   (* Globals changed: *)
   
   
   (************ insert dutys here ***************)
   
   
   (* P00X - Douglas Rd. pumps duty *)
   
   (* set up the the inputs *)
   P00x.qty_motors := 2;
   P00x.bumpless := 0;
   P00x.motor_available := 0;
   motor_available := 0;
   P00x.motor_running := 0;
   
   If P001.remote And P001.auto And P001.permit And Not P001_FL.raw Then
       P00x.motor_available.0 := 1;
   	motor_available := motor_available + 1;
   END_IF;
   If P002.remote And P002.auto And P002.permit And Not P002_FL.raw Then
       P00x.motor_available.1 := 1;
   	motor_available := motor_available + 1;
   END_IF;
   
   If P001.run_sts Then
       P00x.motor_running.0 := 1;
   END_IF;
   If P002.run_sts Then
       P00x.motor_running.1 := 1;
   END_IF;
   
   P00xXA1.raw := motor_available < P00x.qty_motors;
   P00xXA2.raw := motor_available < (P00x.qty_motors - 1);
   
   (* do the duty and reset the momentaries *)
   JSR( DutyRoutine, 1, P00x, P00x );
   
   
   (* flag that powerup is done *)
   duty_pwrup_done := 1;
   
END_ROUTINE

ROUTINE DutyRoutine   (* structured text *)
   SBR( duty );
   
   (* Duty function block *)
   
   (* Does all processing for duty control *)
   
   (* Calling parameters: *)
   (*     duty : DUTY *)
   
   (* Globals used: *)
   
   (* Globals changed: *)
   
   (*-------------------------------------------------------------------------------------------------------------------------------------------------*)
   
   
   (* make the lead motor number legal (in bounds) *)
   IF duty.lead_motor < 1 or duty.lead_motor > duty.qty_motors THEN
       duty.lead_motor := 1;
   END_IF;
   
   (* if the lead motor is selected outside of this subroutine (hard_lead <> 0) *)
   (* set the lead motor to be equal to the hard_lead *)
   IF duty.hard_lead > 0 AND duty.hard_lead <= duty.qty_motors THEN
       duty.lead_motor := duty.hard_lead;
   END_IF;
   
   (* initialise the internal starting parameters *)
   current_motor_index := duty.lead_motor - 1;
   motors_required := duty.motors_required;
   actual_lead_satisfied := 0;
   
   (* loop through each motor starting with the lead, starting or stopping as required and checking runtime *)
   REPEAT
   
   	(* if the motor is unavailable or no more are required, turn off it's output *)
   	IF NOT duty.motor_available.[ current_motor_index ] OR motors_required < 1 THEN
   	    duty.motor_out.[ current_motor_index ] := 0;
   		duty.lead_motor_act := 0;
   
   	(* otherwise turn on its output and decrement the number required *)
   	ELSE
   		duty.motor_out.[ current_motor_index ] := 1;
   		motors_required := motors_required - 1;
   		IF NOT actual_lead_satisfied THEN
   			duty.lead_motor_act := current_motor_index + 1;
   			actual_lead_satisfied := 1;
   		END_IF;
   	END_IF;
   
   	IF motors_required < 1 THEN
   		motors_required := 0;
   	END_IF;
   
   	(* set to the next motor *)
   	current_motor_index := current_motor_index + 1;
   	IF current_motor_index >= duty.qty_motors THEN
   	    current_motor_index := 0;
   	END_IF;
   
   UNTIL current_motor_index = duty.lead_motor - 1
   END_REPEAT;
   
   (* bumpless logic.  Prevents previous motors from shutting off until new requested motors are running *)
   duty.motor_out_want := duty.motor_out;
   duty.motor_out_had := (duty.motor_out_had AND duty.motor_available); (* pump must be available to be allowed to keep running *)
   If duty.bumpless THEN
   	IF duty.motor_out_want <> duty.motor_out_had THEN
   		motors_wanted_running := duty.motor_running AND duty.motor_out_want;
   		IF motors_wanted_running = duty.motor_out_want THEN
   			duty.motor_out_had := motors_wanted_running;
   		ELSIF duty.motors_required < 1 THEN (* If required number of motors to run is zero, set wanted and had motors to 0 *)
   			duty.motor_out_had := 0;
   			duty.motor_out_want := 0;
   		ELSE
   			duty.motor_out := (duty.motor_out_had OR duty.motor_out_want);
   		END_IF;
   	END_IF;
   ELSE
   	duty.motor_out_had := duty.motor_out;
   	duty.motor_out_want := duty.motor_out;
   END_IF;
   
   
   (* now save the unsatisfied counter *)
   duty.unsatisfied_count := motors_required;
   
   (* now process duty rotation *)
   
   if(duty.motors_required=0) then
   	duty.all_motors_stopped.InputBit := 1;
   else
   	duty.all_motors_stopped.InputBit := 0;
   end_if;
   
   (* check for all motors just stopped *)
   OSRI( duty.all_motors_stopped );
   
   (* check for time of day rotation *)
   //IF duty.rotate_interval <= 0 THEN
   //	duty.rotate_interval := 1;
   //END_IF;
   
   GSV(WALLCLOCKTIME,,LocalDateTime, date[0] );
   hour_current := date[ 3 ];
   
   (* New rotation logic to allow rotate on interval of hours rather than days *)
   IF (duty.rotate_hour <> duty.rotate_hour_last) THEN   (* if rotate hour just changed or .. then reset the day and hour offsets *)
   	duty.day_offset := 0;
   	duty.hour_offset := 0;
   	duty.rotated_today := 0;
   ELSIF (hour_current < duty.hour_last) THEN (* if the day just changed, calculate a new hour offset *)
   	duty.day_offset := duty.day_offset + 1;
   	duty.hour_offset := duty.day_offset * (24 MOD duty.rotate_hour);
   END_IF;
   IF hour_current <> duty.hour_last THEN duty.rotated_today := 0; END_IF;
   duty.rotate_hour_last := duty.rotate_hour;
   duty.hour_last := hour_current;
   
   //duty.date_os.InputBit := date[ 3 ] = duty.rotate_hour;
   //OSRI( duty.date_os );
   //IF duty.date_os.OutputBit THEN
   //    duty.rotate_daycount := duty.rotate_daycount + 1;
   //END_IF;
   
   
   
   (* finally, rotate if required and lead is not 'hard' *)
   IF duty.hard_lead < 1 THEN
   
   	(* First check if we hit the daycount *)
   	IF ((hour_current = duty.rotate_hour) AND NOT duty.rotated_today) THEN
   		duty.rotate_daycount := duty.rotate_daycount + 1;
   	END_IF;
   	IF
   			(* Rotate on Stop *)
   	        (duty.all_motors_stopped.OutputBit AND duty.rotate_on_stop)
   	    OR
   			(* Rotate on time - time of day *)
   		    ((duty.rotate_daycount >= duty.rotate_interval) AND duty.rotate_on_time AND (hour_current = duty.rotate_hour) AND NOT duty.rotated_today AND (duty.rotate_interval > 0))
   		OR
   			(* Rotate on time - every so many hours *)
   		    ((((hour_current + duty.hour_offset) MOD duty.rotate_hour) = 0) AND duty.rotate_on_time AND NOT duty.rotated_today AND (duty.rotate_interval = 0))
   		OR
   			(* Rotate manual *)
   		    duty.rotate_man
   	THEN
   
   		(* rotate until there is a motor that is available *)
   		current_motor_index := duty.lead_motor - 1;
   		REPEAT
   		    current_motor_index := current_motor_index + 1;
   			IF current_motor_index >= duty.qty_motors THEN
   		        current_motor_index := 0;
   		    END_IF;
   		UNTIL duty.motor_available.[ current_motor_index ] OR current_motor_index = duty.lead_motor - 1 //OR duty.rotate_man
   		END_REPEAT;
   		duty.rotate_daycount := 0;
   		duty.lead_motor := current_motor_index + 1;
   
   
   		(* if it's midnight and we've just rotated then reset the day / hour offset to 0 (ie if the cycle is starting over) *)
   		IF ((((hour_current + duty.hour_offset) MOD duty.rotate_hour) = 0) AND (hour_current = 0)) THEN
   			duty.day_offset := 0;
   			duty.hour_offset := 0;
   		END_IF;
   
   		(* prevent multiple rotations per hour *)
   		duty.rotated_today := 1;
   
   	END_IF;
   END_IF;
   
   (* turn off the momentary rotate *)
   IF duty.rotate_man THEN duty.rotate_man := 0; END_IF;
   
   RET( duty );
   
END_ROUTINE
END_PROGRAM

PROGRAM FaultProgram   (* main routine FaultRoutine *)
VAR
   major_fault : FAULTRECORD := (time_low := 2139313344, time_high := 210899, info[0] := 16#0000_0001, info[1] := 16#0000_2420, info[2] := 16#0000_0203);
   major_fault_code_last : INT := 16;
   major_fault_type_last : INT := 3;
END_VAR

ROUTINE FaultRoutine   (* structured text *)
   (* Fault processing program *)
   
   (* Does all basic processing for processor faults *)
   
   (* Globals used: *)
   
   (* Globals changed: *)
   
   (*-------------------------------------------------------------------------------------------------------------------------------------------------*)
   
   
   (* get the fault record *)
   GSV( PROGRAM, THIS, MAJORFAULTRECORD, major_fault.time_low );
   
   (* clear the fault *)
   major_fault_type_last := major_fault.type;
   major_fault.type := 0;
   major_fault_code_last := major_fault.code;
   major_fault.code := 0;
   
   (* return the fault record *)
   SSV( PROGRAM, THIS, MAJORFAULTRECORD, major_fault.time_low );
   
END_ROUTINE
END_PROGRAM

PROGRAM FunctionBlockInit   (* main routine Init *)
VAR
   major_fault : FAULTRECORD := (time_low := -1970702789, time_high := 381732, info[0] := 16#671b_9f6b, info[1] := 16#0005_d323);
END_VAR

ROUTINE Init   (* structured text *)
   (* powerup initialisation *)
   
   (* flag that powerup must be done in the individual programs *)
   main_comm_pwrup_done := 0;
   motor_pwrup_done := 0;
   valve_pwrup_done := 0;
   analogfb_pwrup_done := 0;
   digitalnf_pwrup_done := 0;
   alm_pwrup_done := 0;
   pranalog_pwrup_done := 0;
   pid_pwrup_done := 0;
   duty_pwrup_done := 0;
   sequence_pwrup_done := 0;
   report_pwrup_done := 0;
   
   (* get the fault record *)
   GSV( PROGRAM, THIS, MAJORFAULTRECORD, major_fault.time_low );
   
   (* clear the fault *)
   major_fault.type := 0;
   major_fault.code := 0;
   
   (* return the fault record *)
   SSV( PROGRAM, THIS, MAJORFAULTRECORD, major_fault.time_low );
   
END_ROUTINE
END_PROGRAM

PROGRAM Inputs   (* main routine Inputs *)

ROUTINE Inputs   (* structured text *)
   (* copy i/o into tags *)
   
   (* Slot 1 8AI *)
   FIT001.raw := (Local:1:I.Ch0Data - 4000) / 16000 * 100;
   LIT001.raw := (Local:1:I.Ch1Data - 4000) / 16000 * 100;
   // := (Local:1:I.Ch2Data - 4000) / 16000 * 100;
   // := (Local:1:I.Ch3Data - 4000) / 16000 * 100;
   
   (* Slot 2 16DI *)
   P001.remote := Local:2:I.Data.0 AND NOT XAFLOAT.raw;
   P001.run_sts := Local:2:I.Data.1;
   P001_OL := Local:2:I.Data.2;
   P001_TMP := Local:2:I.Data.3;
   P001_LK := Local:2:I.Data.4;
   P002.remote := Local:2:I.Data.5 AND NOT XAFLOAT.raw;
   P002.run_sts := Local:2:I.Data.6;
   P002_OL := Local:2:I.Data.7;
   P002_TMP := Local:2:I.Data.8;
   P002_LK := Local:2:I.Data.9;
   CRP.raw := Local:2:I.Data.10;
   LSH001.raw := Local:2:I.Data.11;
   LSH002.raw := Local:2:I.Data.12;
   XAFLOAT.raw := Local:2:I.Data.13;
   // := Local:2:I.Data.14;
   // := Local:2:I.Data.15;
   
   (* Slot 3 16DI *)
   P00x.hard_lead.0 := Local:3:I.Data.0;
   P00x.hard_lead.1 := Local:3:I.Data.1;
   ALM_RESET := Local:3:I.Data.2;
   ALM_TEST := Local:3:I.Data.3;
   ALM_ACK := Local:3:I.Data.4;
   DG1LSL1.raw := Local:3:I.Data.5;
   DG1LSL2.raw := Local:3:I.Data.6;
   DG1BAT.raw := Local:3:I.Data.7;
   DG1.run_sts := Local:3:I.Data.8;
   DG1_FL.raw := Local:3:I.Data.9;
   ATSGEN.raw := Local:3:I.Data.10;
   ATSFLT.raw := Local:3:I.Data.11;
   // := Local:3:I.Data.12;
   // := Local:3:I.Data.13;
   // := Local:3:I.Data.14;
   // := NOT Local:3:I.Data.15;
   
END_ROUTINE
END_PROGRAM

PROGRAM LevelBandControl   (* main routine LevelBandControl *)
VAR
   controllevel : REAL := 0.9637501;
   pump_speed : REAL;
END_VAR

ROUTINE LevelBandControl   (* structured text *)
   (* simple band control *)
   controllevel := LIT001.value;
   
   
   (* set band *)
   CASE BAND_CURRENT OF
   
   0:
   	IF controllevel > BAND_B01_START THEN
   		BAND_CURRENT := 1;
   	END_IF;
   
   1:
   	IF controllevel < BAND_B01_STOP THEN
   		BAND_CURRENT := 0;
   	ELSIF controllevel > BAND_B02_START THEN
   		BAND_CURRENT := 2;
   	END_IF;
   
   2:
   	IF controllevel < BAND_B02_STOP THEN
   		BAND_CURRENT := 1;
   	END_IF;
   
   ELSE
   	BAND_CURRENT := 0;
   END_CASE;
   
   
   (* set speed *)
   CASE BAND_CURRENT OF
   
   0:
   	pump_speed := 0;
   
   1:
   	IF controllevel < BAND_B01_MINSPD_LVL THEN
   		pump_speed := 0;
   	ELSIF controllevel > BAND_B01_MAXSPD_LVL THEN
   		pump_speed := 100;
   	ELSE
   		pump_speed := (controllevel - BAND_B01_MINSPD_LVL) / (BAND_B01_MAXSPD_LVL - BAND_B01_MINSPD_LVL) * 100;
   	END_IF;
   
   2:
   	IF controllevel < BAND_B02_MINSPD_LVL THEN
   		pump_speed := 0;
   	ELSIF controllevel > BAND_B02_MAXSPD_LVL THEN
   		pump_speed := 100;
   	ELSE
   		pump_speed := (controllevel - BAND_B02_MINSPD_LVL) / (BAND_B02_MAXSPD_LVL - BAND_B02_MINSPD_LVL) * 100;
   	END_IF;
   
   END_CASE;
   
   
   (* run pumps *)
   P00x.motors_required := BAND_CURRENT;
   P001.start_auto := P00x.motor_out.0;
   P001.stop_auto := NOT P00x.motor_out.0;
   P002.start_auto := P00x.motor_out.1;
   P002.stop_auto := NOT P00x.motor_out.1;
   IF P001.run_sts THEN
   	P001SP.out_auto := pump_speed;
   ELSE
   	P001SP.out_auto := 0;
   END_IF;
   IF P002.run_sts THEN
   	P002SP.out_auto := pump_speed;
   ELSE
   	P002SP.out_auto := 0;
   END_IF;
   
END_ROUTINE
END_PROGRAM

PROGRAM MotorProgram   (* main routine Motors *)
VAR
   fail_pending : BOOL;
   motor : MOTOR := (fail_dlay := 60, auto := 1, remote := 1, permit := 1, stop_sts := 1, runtime := 0.0011108334, runtime_f := 0.0011108334, fail_tonr.TimerEnable := 1, fail_tonr.PRE := 60000, fail_tonr.Reset := 1, manual_mode_timer.Reset := 1);
   permit_start : BOOL := 1;
   pwrup_dlayd : FBD_TIMER := (TimerEnable := 1, PRE := 10000, ACC := 10000, EN := 1, DN := 1);
   start_dlayd : FBD_TIMER := (TimerEnable := 1, PRE := 10, ACC := 250, EN := 1, DN := 1);
   start_permit : BOOL := 1;
END_VAR

ROUTINE MotorRoutine   (* structured text *)
   SBR(motor, permit_start);
   
   (* Motor function block *)
   
   (* Does all motor control processing *)
   
   (* Calling parameters: *)
   (*     motor : MOTOR *)
   (*     permit_start : BOOL start allowed *)
   
   (* Globals used: *)
   (*     pwrup_dlayd *)
   (*     functionblocktask_cycle_time *)
   
   (* Globals changed: *)
   (*     fail_pending *)
   
   (*-------------------------------------------------------------------------------------------------------------------------------------------------*)
   
   
   (* Load fault time with preset value *)
   motor.fail_tonr.PRE := motor.fail_dlay * 1000;
   
   
   (* handle the failure logic first *)
   
   (* calculate the fail pending *)
   IF
           NOT motor.remote
       OR
           ( motor.run_out AND motor.run_sts AND NOT motor.stop_sts )
       OR
           ( NOT motor.run_out AND NOT motor.run_sts AND motor.stop_sts )
   	OR
   	    NOT pwrup_dlayd.DN
   	OR
   		motor.fail_reset
   THEN
       fail_pending := 0;
   ELSE
       fail_pending := 1;
   END_IF;
   
   (* time the fail pending *)
   motor.fail_tonr.TimerEnable := 1;
   motor.fail_tonr.Reset := NOT fail_pending;
   motor.manual_mode_timer.PRE := motor.mode_dlay * 1000 *60;
   
   (*If motor is in  manual mode and time greater then 0 then allow tiemr to revert to auto automatically*)
   motor.manual_mode_timer.Reset := motor.auto or (motor.mode_dlay = 0);
   
   TONR(motor.fail_tonr);
   
   TONR(motor.manual_mode_timer);
   //revert to auto
   if motor.manual_mode_timer.DN then
   	motor.auto := 1;
   end_if;
   
   (* calculate the fail and clear if we're not in remote or if we just powered up *)
   motor.fail := ( motor.fail AND ( NOT motor.fail_reset AND motor.remote AND pwrup_dlayd.DN ) ) OR motor.fail_tonr.DN;
   
   
   (* handle the motor desired state and outputs *)
   
   (* if we're failed or not permitted to run, set desired state to stopped *)
   IF motor.fail OR NOT motor.permit THEN
       motor.run_out := 0;
   
   (* if not in auto process the manual commands *)
   ELSIF NOT motor.auto THEN
       motor.run_out := ( motor.run_out OR ( motor.start_man AND permit_start ) ) AND NOT motor.stop_man;
   
   (* finally process the auto commands *)
   ELSE
       motor.run_out := ( motor.run_out OR ( motor.start_auto AND permit_start ) ) AND NOT motor.stop_auto;
   END_IF;
   
   (* create the motor outputs - only energize if we're in remote *)
   IF motor.remote THEN
   	motor.stop_out := NOT motor.run_out AND ( motor.run_sts OR NOT motor.stop_sts );
   	motor.start_out := motor.run_out AND ( NOT motor.run_sts OR motor.stop_sts );
   ELSE
   	motor.stop_out := 0;
   	motor.start_out := 0;
   END_IF;
   
   
   (* check for just starting *)
   motor.start_os.InputBit := motor.run_out;
   OSRI(motor.start_os);
   
   
   (* accumulate runtime modulo 1e5 *)
   
   (* if we're running, add on the cycle time *)
   IF motor.run_sts THEN
   
       (* add the cycle time to the fractional part *)
       motor.runtime_f := motor.runtime_f + FunctionBlock_Cycle_Time / 1000.0 / 3600.0;
   
       (* make sure the fractional part is <1 *)
   	WHILE motor.runtime_f >= 1.0 DO
   	    motor.runtime_i := motor.runtime_i + 1;
   		motor.runtime_f := motor.runtime_f - 1;
   	END_WHILE;
   
       (* make the runtime modulo 1e6 *)
       WHILE motor.runtime_i >= 100000.0 DO
           motor.runtime_i := motor.runtime_i - 100000;
       END_WHILE;
   
   	(* combine two parts to make runtime *)
   	motor.runtime := motor.runtime_f + motor.runtime_i;
   
   END_IF;
   
   (* reset the momentary pushbuttons *)
   
   (* reset the momentary inputs *)
    IF  motor.stop_man THEN  motor.stop_man := 0; END_IF;
    IF  motor.start_man THEN  motor.start_man := 0; END_IF;
    IF  motor.stop_auto THEN  motor.stop_auto := 0; END_IF;
    IF  motor.start_auto THEN  motor.start_auto := 0; END_IF;
    IF  motor.fail_reset THEN  motor.fail_reset := 0; END_IF;
   
   motor.Gen_Alarm := motor.fail;
   ret(motor);
   
END_ROUTINE

ROUTINE Motors   (* structured text *)
   (* Motor processing program *)
   
   (* Does all basic processing for all motors by setting up inputs then calling the motor function block for each *)
   
   (* Globals used: *)
   
   (* Globals changed: *)
   (*     motor_pwrup_done *)
   (*     pwrup_dlayd *)
   (*     cycle_time *)
   (*     each motor *)
   
   (*-------------------------------------------------------------------------------------------------------------------------------------------------*)
   
   
   (* use a TONR to delay power recovery *)
   
   pwrup_dlayd.Reset := not motor_pwrup_done;
   TONR(pwrup_dlayd);
   
   
   (* time the start delay (note: remove any reset from last execution *)
   TONR(start_dlayd);
   start_dlayd.Reset := 0;
   
   
   (* process each motor as follows: (note these comments are only shown here for brevity) *)
   (*     1. set up inputs (specific to each motor and commented *)
   (*     2. call the motor processing function block *)
   (*     3. clear the momentary inputs if they were on *)
   (*     4. set up the start delay timer if we just started *)
   (*     5. get the outputs *)
   
   
   (************ insert motors here ***************)
   
   
   
   
   (* P001 Raw sewage pump 1 *)
   
   (* set up the inputs *)
   
   P001.permit := NOT CRP.raw AND NOT P001_OL AND NOT P001_LK AND NOT P001_TMP; //Power and not Overload and not Leak and not Temp
   
   P001.stop_sts := NOT P001.run_sts;
   
   (* process the motor and adjust the start delay if required*)
   start_permit := P001.start_dlay = 0 OR start_dlayd.DN;
   JSR( MotorRoutine, 2, P001, start_permit, P001 );
   IF (P001.start_os.OutputBit AND (P001.start_dlay > 0)) THEN
       start_dlayd.PRE := P001.start_dlay;
       start_dlayd.Reset := 1;
       TONR(start_dlayd);
   END_IF;
   P001_FL.raw := P001.fail OR P001_OL OR P001_LK OR P001_TMP;
   
   
   (* P002 Raw sewage pump 2 *)
   
   (* set up the inputs *)
   
   P002.permit := NOT CRP.raw AND NOT P002_OL AND NOT P002_LK AND NOT P002_TMP; //Power and not Overload and not Leak and not Temp
   
   P002.stop_sts := NOT P002.run_sts;
   
   (* process the motor and adjust the start delay if required*)
   start_permit := P002.start_dlay = 0 OR start_dlayd.DN;
   JSR( MotorRoutine, 2, P002, start_permit, P002 );
   IF (P002.start_os.OutputBit AND (P002.start_dlay > 0)) THEN
       start_dlayd.PRE := P002.start_dlay;
       start_dlayd.Reset := 1;
       TONR(start_dlayd);
   END_IF;
   P002_FL.raw := P002.fail OR P002_OL OR P002_LK OR P002_TMP;
   
   
   (* DG1 Diesel generator *)
   
   (* set up the inputs *)
   DG1.remote := NOT DG1.fail;
   DG1.permit := 1; //n/a no control
   
   DG1.stop_sts := NOT DG1.run_sts;
   (* simulate the commands to keep the screen clean *)
   DG1.auto := 1;
   DG1.start_auto := DG1.run_sts;
   DG1.stop_auto := DG1.stop_sts;
   DG1.fail_dlay := 60;
   
   (* process the motor and adjust the start delay if required*)
   start_permit := DG1.start_dlay = 0 OR start_dlayd.DN;
   JSR( MotorRoutine, 2, DG1, start_permit, DG1 );
   IF (DG1.start_os.OutputBit AND (DG1.start_dlay > 0)) THEN
       start_dlayd.PRE := DG1.start_dlay;
       start_dlayd.Reset := 1;
       TONR(start_dlayd);
   END_IF;
   //DG1_FL.raw := DG1.fail; taken from input general fault instead
   
   
   
   (* flag that powerup is done *)
   motor_pwrup_done := 1;
   
END_ROUTINE
END_PROGRAM

PROGRAM Notes   (* main routine Rev_Notes *)

ROUTINE Rev_Notes   (* structured text *)
   (*
   
   June 24, 2010 MS  Added BWQUEUE user-defined datatype
   June 24, 2010 MS  Added CT user-defined datatype
   June 24, 2010 MS  Added check for NAN logic to Pranalog_Routine
   June 24, 2010 MS  Added check for NAN logic to Report routines (5, 15, standard)
   June 24, 2010 MS  Prevent motor maintained outputs from energizing when not remote
   June 24, 2010 MS  Add log delete routine to report routines (5, 15, standard)
   June 24, 2010 MS  Change report data routines so that 0 is 'duration' and motors start at 1
   July 21, 2010 KL  Changed program Notes (in Unscheduled Programs task) to have main routine Rev_Notes to avoid warning during verify
   
   *)
END_ROUTINE
END_PROGRAM

PROGRAM Outputs   (* main routine Outputs *)

ROUTINE Outputs   (* structured text *)
   (* put i/o here *)
   
   
   
   (* Slot 4 16DO *)
   Local:4:O.Data.0 := NOT P001.permit;
   Local:4:O.Data.1 := P001.run_out;
   Local:4:O.Data.2 := Dialer[0];			//P001_FL.chan := 1;
   Local:4:O.Data.3 := NOT P002.permit;
   Local:4:O.Data.4 := P002.run_out;
   Local:4:O.Data.5 := Dialer[1];			//P002_FL.chan := 2;
   Local:4:O.Data.6 := Dialer[4];			//LIT001_FL.chan := 5;
   Local:4:O.Data.7 := Dialer[2];			//LIT001_hh.chan := 3;  LSH002.chan := 3; LSH001.chan := 3;
   Local:4:O.Data.8 := Dialer[3];			//LIT001_ll.chan := 4;
   Local:4:O.Data.9 := Dialer[5];			//XAFLOAT.chan := 6;
   Local:4:O.Data.10 := Dialer[6];			//ATSGEN.chan := 7;
   Local:4:O.Data.11 := Dialer[7];			//ATSFLT.chan := 8;
   Local:4:O.Data.12 := Dialer[8];			//DG1_FL.chan := 9;
   Local:4:O.Data.13 := Dialer[9];			//DG1RUN.chan := 10;
   Local:4:O.Data.14 := Dialer[10];		//DG1LSL1.chan := 11;
   Local:4:O.Data.15 := Dialer[11];		//DG1LSL2.chan := 12;
   
   (* Slot 5 8DO *)
   Local:5:O.Data.0 := Dialer[12];			//DG1BAT.chan := 13;
   Local:5:O.Data.1 := DIALOUT_ON;
   Local:5:O.Data.2 := DIALOUT_ON;
   Local:5:O.Data.3 := 0;
   Local:5:O.Data.4 := 0;
   Local:5:O.Data.5 := 0;
   Local:5:O.Data.6 := 0;
   Local:5:O.Data.7 := 0;
   
END_ROUTINE
END_PROGRAM

PROGRAM PIDProgram   (* main routine PIDs *)
VAR
   out_temp : REAL;
   pid_controller : PIDBLOCK := (PV_MaxEU := 500.0, FLOW_MaxEU := 100.0, AUTO := 1, KP := 0.5, KI := 5.0, FORCE := 1, embeddedPID.CTL := -1980725376, embeddedPID.EN := 1, embeddedPID.DOE := 1, embeddedPID.MO := 1, embeddedPID.PE := 1, embeddedPID.NDF := 1, embeddedPID.NOBC := 1, embeddedPID.NOZC := 1, embeddedPID.INI := 1, embeddedPID.DVNA := 1, embeddedPID.DVPA := 1, embeddedPID.PVLA := 1, embeddedPID.PVHA := 1, embeddedPID.KP := 0.5, embeddedPID.KI := 0.2, embeddedPID.MAXS := 100.0, embeddedPID.MAXO := 100.0, embeddedPID.UPD := 0.25, embeddedPID.MAXI := 100.0, embeddedPID.MAXCV := 100.0, embeddedPID.MAXTIE := 100.0, embeddedPID.DATA[5] := 1.0, embeddedPID.DATA[6] := 1.0, embeddedPID.DATA[7] := 4.0, embeddedPID.DATA[8] := 0.5, embeddedPID.DATA[9] := 0.2, embeddedPID.DATA[11] := 0.5, embeddedPID.DATA[12] := 0.041666668, embeddedPID.DATA[15] := 1.0, embeddedPID.DATA[16] := 1.0);
   tieback : REAL;
END_VAR

ROUTINE PIDRoutine   (* structured text *)
   SBR(pid_controller);
   
   (* PID control function block *)
   
   (* Does all PID control processing *)
   
   (* Calling parameters: *)
   (*     pid_controller : PIDBLOCK *)
   
   (* Globals used: *)
   (*     pwrup_dlayd *)
   (*     cycle_time *)
   
   (* Globals changed: *)
   
   (*-------------------------------------------------------------------------------------------------------------------------------------------------*)
   
   (* set up the PID configurations *)
   pid_controller.embeddedPID.MAXS := 100;
   pid_controller.embeddedPID.MINS := 0;
   pid_controller.embeddedPID.MAXO := 100;
   pid_controller.embeddedPID.MINO := 0;
   pid_controller.embeddedPID.MAXI := 100;
   pid_controller.embeddedPID.MINI := 0;
   pid_controller.embeddedPID.MAXCV := 100;
   pid_controller.embeddedPID.MINCV := 0;
   pid_controller.embeddedPID.MAXTIE := 100;
   pid_controller.embeddedPID.MINTIE := 0;
   pid_controller.embeddedPID.UPD := 0.25;
   pid_controller.embeddedPID.EN := 1;
   pid_controller.embeddedPID.DOE := 1;
   pid_controller.embeddedPID.PE := 1;
   pid_controller.embeddedPID.NDF := 1;
   pid_controller.embeddedPID.NOBC := 1;
   pid_controller.embeddedPID.NOZC := 1;
   pid_controller.embeddedPID.SWM := 0;
   
   (* copy appropriate stuff into the embedded PID *)
   pid_controller.PV_PCT := (pid_controller.PV - pid_controller.PV_MinEU) / (pid_controller.PV_MaxEU - pid_controller.PV_MinEU) * 100;
   pid_controller.SP_PCT := (pid_controller.SP - pid_controller.PV_MinEU) / (pid_controller.PV_MaxEU - pid_controller.PV_MinEU) * 100;
   pid_controller.FLOW_PCT := (pid_controller.FLOW - pid_controller.FLOW_MinEU) / (pid_controller.FLOW_MaxEU - pid_controller.FLOW_MinEU) * 100;
   
   
   IF pid_controller.KP < 0 THEN
   	pid_controller.embeddedPID.CA := 1;
   	pid_controller.embeddedPID.KP := 0-pid_controller.KP;
   ELSE
   	pid_controller.embeddedPID.CA := 0;
   	pid_controller.embeddedPID.KP := pid_controller.KP;
   END_IF;
   IF pid_controller.KI > 0 THEN
   	pid_controller.embeddedPID.KI := 1/pid_controller.KI;
   ELSE
   	pid_controller.embeddedPID.KI :=0;
   END_IF;
   pid_controller.embeddedPID.KD := pid_controller.KD;
   pid_controller.embeddedPID.SP := pid_controller.SP_PCT;
   
   (* if we're in manual, set the output to the operator value *)
   IF NOT pid_controller.AUTO THEN
       pid_controller.embeddedPID.MO := 1;
   	tieback := pid_controller.OUT_MAN;
   
   (* if the output is forced, set the output *)
   ELSIF pid_controller.FORCE THEN
       pid_controller.embeddedPID.MO := 1;
   	tieback := pid_controller.FORCE_VALUE;
   
   (* if we're compound and either no flow or 100% on final output, freeze PID *)
   ELSIF
   		pid_controller.MODE
   	AND
   		(
   			(pid_controller.FLOW = 0)
   		OR
   			(
   				((pid_controller.OUT * pid_controller.K / 2 * pid_controller.FLOW_PCT / 10000) > 100)
   			AND
   				(
   					((pid_controller.PV > pid_controller.SP) AND (pid_controller.KP > 0))
   				OR
   					((pid_controller.PV < pid_controller.SP) AND (pid_controller.KP < 0))
   				)
   			)
   		)
   THEN
       pid_controller.embeddedPID.MO := 1;
   	tieback := pid_controller.OUT;
   
   (* otherwise, let the PID work *)
   ELSE
       pid_controller.embeddedPID.MO := 0;
   END_IF;
   
   (* execute the PID *)
   PID( pid_controller.embeddedPID, pid_controller.PV_PCT, tieback, pid_controller.OUT, 0, 0, 0 );
   
   (* make the output *)
   IF pid_controller.MODE THEN
   	out_temp := pid_controller.OUT / 100 * pid_controller.K * 2 * pid_controller.FLOW_PCT / 100;
   	IF out_temp > 100 THEN
   		pid_controller.OUT := 100;
   	ELSIF out_temp < 0 THEN
   		pid_controller.OUT := 0;
   	ELSE
   		pid_controller.FinalOut := out_temp;
   	END_IF;
   ELSE
   	pid_controller.FinalOut := pid_controller.OUT;
   END_IF;
   
   (* finally, prepare for bumpless from auto to man *)
   IF pid_controller.AUTO THEN
   	pid_controller.OUT_MAN := pid_controller.OUT ;
   END_IF;
   
   ret(pid_controller);
   
END_ROUTINE

ROUTINE PIDs   (* structured text *)
   (* PID controllers function block *)
   
   (* Does processing for each PID controller *)
   
   (* Calling parameters: *)
   
   (* Globals used: *)
   
   (* Globals changed: *)
   
   (*-------------------------------------------------------------------------------------------------------------------------------------------------*)
   
   
   (************ insert PIDs here ***************)
   
   
   (* flag that powerup is done *)
   pid_pwrup_done := 1;
   
END_ROUTINE
END_PROGRAM
